(* IEC 61131-3 sources: RL_MAR/experiments/comparison/llm4plc/results/gpt-4o-mini_20260506_100619/20260506_101408, 3 files *)

(* ---- generated_code_iteration_0.st ---- *)
ructured-text
FUNCTION_BLOCK FB_SplitNumber
VAR_INPUT
    InputNumber : INT;
END_VAR

VAR_OUTPUT
    Thousands : INT;
    Hundreds : INT;
    Tens : INT;
    Ones : INT;
    Min : INT;
    error : BOOL;
    status : WORD;
END_VAR

VAR
    state : INT; // THE STATE VARIABLE
    prevState : INT; // THE PREVIOUS STATE VARIABLE
    tempNumber : INT; // Temporary variable for processing
    minValue : INT; // Variable to track the minimum non-zero digit
END_VAR

// Initialize state
state := 0;
error := FALSE;
status := 16#0000;
Thousands := 0;
Hundreds := 0;
Tens := 0;
Ones := 0;
Min := 0;

CASE state OF
    0: // STATE 0: INITIALIZE
        // Always transition to validate input
        state := 1;

    1: // STATE 1: VALIDATE INPUT
        IF InputNumber < 0 OR InputNumber > 9999 THEN
            error := TRUE;
            status := 16#8001;
            Thousands := 0;
            Hundreds := 0;
            Tens := 0;
            Ones := 0;
            Min := 0;
            state := 4; // Transition to ERROR HANDLING
        ELSE
            error := FALSE;
            status := 16#0000;
            state := 2; // Transition to SEPARATE DIGITS
        END_IF;

    2: // STATE 2: SEPARATE DIGITS
        Thousands := InputNumber / 1000;
        Hundreds := (InputNumber MOD 1000) / 100;
        Tens := (InputNumber MOD 100) / 10;
        Ones := InputNumber MOD 10;
        Min := 0; // Initialize Min
        state := 3; // Transition to FIND MINIMUM NON-ZERO DIGIT

    3: // STATE 3: FIND MINIMUM NON-ZERO DIGIT
        minValue := 32767; // Initialize minValue to maximum possible INT value

        // Compare non-zero digits
        IF Thousands > 0 THEN
            minValue := minimal(minValue, Thousands);
        END_IF;

        IF Hundreds > 0 THEN
            minValue := minimal(minValue, Hundreds);
        END_IF;

        IF Tens > 0 THEN
            minValue := minimal(minValue, Tens);
        END_IF;

        IF Ones > 0 THEN
            minValue := minimal(minValue, Ones);
        END_IF;

        // Set Min based on minValue
        IF minValue = 32767 THEN
            Min := 0; // All digits were zero
        ELSE
            Min := minValue; // Found minimum non-zero digit
        END_IF;

        state := 0; // Transition back to INITIALIZE

    4: // STATE 4: ERROR HANDLING
        // Error state already handled in STATE 1
        state := 0; // Transition back to INITIALIZE
END_CASE;

END_FUNCTION_BLOCK

(* ---- generated_code_iteration_1.st ---- *)
START_REASON
The errors in the original Structured Text (ST) code were primarily due to the incorrect handling of variable declarations and the use of the variable name "Min." In ST, "Min" is a reserved keyword in some contexts, which can lead to unexpected behavior or compilation errors. To resolve this, I will rename the variable "Min" to "MinimumValue" to avoid any conflicts. Additionally, I will ensure that the variable sections are correctly closed with "END_VAR" as required.
END_REASON

START_ST
FUNCTION_BLOCK FB_SplitNumber
VAR_INPUT
    InputNumber : INT;
END_VAR

VAR_OUTPUT
    Thousands : INT;
    Hundreds : INT;
    Tens : INT;
    Ones : INT;
    MinimumValue : INT; // Renamed from Min to MinimumValue
    error : BOOL;
    status : WORD;
END_VAR

VAR
    state : INT; // THE STATE VARIABLE
    prevState : INT; // THE PREVIOUS STATE VARIABLE
    tempNumber : INT; // Temporary variable for processing
    minValue : INT; // Variable to track the minimum non-zero digit
END_VAR

// Initialize state
state := 0;
error := FALSE;
status := 16#0000;
Thousands := 0;
Hundreds := 0;
Tens := 0;
Ones := 0;
MinimumValue := 0; // Initialize MinimumValue

CASE state OF
    0: // STATE 0: INITIALIZE
        // Always transition to validate input
        state := 1;

    1: // STATE 1: VALIDATE INPUT
        IF InputNumber < 0 OR InputNumber > 9999 THEN
            error := TRUE;
            status := 16#8001;
            Thousands := 0;
            Hundreds := 0;
            Tens := 0;
            Ones := 0;
            MinimumValue := 0; // Set MinimumValue to 0 on error
            state := 4; // Transition to ERROR HANDLING
        ELSE
            error := FALSE;
            status := 16#0000;
            state := 2; // Transition to SEPARATE DIGITS
        END_IF;

    2: // STATE 2: SEPARATE DIGITS
        Thousands := InputNumber / 1000;
        Hundreds := (InputNumber MOD 1000) / 100;
        Tens := (InputNumber MOD 100) / 10;
        Ones := InputNumber MOD 10;
        MinimumValue := 0; // Initialize MinimumValue
        state := 3; // Transition to FIND MINIMUM NON-ZERO DIGIT

    3: // STATE 3: FIND MINIMUM NON-ZERO DIGIT
        minValue := 32767; // Initialize minValue to maximum possible INT value

        // Compare non-zero digits
        IF Thousands > 0 THEN
            minValue := minimal(minValue, Thousands);
        END_IF;

        IF Hundreds > 0 THEN
            minValue := minimal(minValue, Hundreds);
        END_IF;

        IF Tens > 0 THEN
            minValue := minimal(minValue, Tens);
        END_IF;

        IF Ones > 0 THEN
            minValue := minimal(minValue, Ones);
        END_IF;

        // Set MinimumValue based on minValue
        IF minValue = 32767 THEN
            MinimumValue := 0; // All digits were zero
        ELSE
            MinimumValue := minValue; // Found minimum non-zero digit
        END_IF;

        state := 0; // Transition back to INITIALIZE

    4: // STATE 4: ERROR HANDLING
        // Error state already handled in STATE 1
        state := 0; // Transition back to INITIALIZE
END_CASE;

END_FUNCTION_BLOCK
END_ST

(* ---- generated_code_iteration_2.st ---- *)
START_REASON
The errors in the original Structured Text (ST) code were primarily due to the incorrect use of the function "minimal." In Structured Text, there is no built-in function named "minimal" for comparing values. Instead, I should use a conditional statement to determine the minimum value among the digits. I will replace the usage of "minimal" with appropriate conditional checks to find the minimum non-zero digit. Additionally, I will ensure that the variable sections are correctly closed with "END_VAR" as required.
END_REASON

START_ST
FUNCTION_BLOCK FB_SplitNumber
VAR_INPUT
    InputNumber : INT;
END_VAR

VAR_OUTPUT
    Thousands : INT;
    Hundreds : INT;
    Tens : INT;
    Ones : INT;
    MinimumValue : INT; // Renamed from Min to MinimumValue
    error : BOOL;
    status : WORD;
END_VAR

VAR
    state : INT; // THE STATE VARIABLE
    prevState : INT; // THE PREVIOUS STATE VARIABLE
    tempNumber : INT; // Temporary variable for processing
    minValue : INT; // Variable to track the minimum non-zero digit
END_VAR

// Initialize state
state := 0;
error := FALSE;
status := 16#0000;
Thousands := 0;
Hundreds := 0;
Tens := 0;
Ones := 0;
MinimumValue := 0; // Initialize MinimumValue

CASE state OF
    0: // STATE 0: INITIALIZE
        // Always transition to validate input
        state := 1;

    1: // STATE 1: VALIDATE INPUT
        IF InputNumber < 0 OR InputNumber > 9999 THEN
            error := TRUE;
            status := 16#8001;
            Thousands := 0;
            Hundreds := 0;
            Tens := 0;
            Ones := 0;
            MinimumValue := 0; // Set MinimumValue to 0 on error
            state := 4; // Transition to ERROR HANDLING
        ELSE
            error := FALSE;
            status := 16#0000;
            state := 2; // Transition to SEPARATE DIGITS
        END_IF;

    2: // STATE 2: SEPARATE DIGITS
        Thousands := InputNumber / 1000;
        Hundreds := (InputNumber MOD 1000) / 100;
        Tens := (InputNumber MOD 100) / 10;
        Ones := InputNumber MOD 10;
        MinimumValue := 0; // Initialize MinimumValue
        state := 3; // Transition to FIND MINIMUM NON-ZERO DIGIT

    3: // STATE 3: FIND MINIMUM NON-ZERO DIGIT
        minValue := 32767; // Initialize minValue to maximum possible INT value

        // Compare non-zero digits
        IF Thousands > 0 AND Thousands < minValue THEN
            minValue := Thousands;
        END_IF;

        IF Hundreds > 0 AND Hundreds < minValue THEN
            minValue := Hundreds;
        END_IF;

        IF Tens > 0 AND Tens < minValue THEN
            minValue := Tens;
        END_IF;

        IF Ones > 0 AND Ones < minValue THEN
            minValue := Ones;
        END_IF;

        // Set MinimumValue based on minValue
        IF minValue = 32767 THEN
            MinimumValue := 0; // All digits were zero
        ELSE
            MinimumValue := minValue; // Found minimum non-zero digit
        END_IF;

        state := 0; // Transition back to INITIALIZE

    4: // STATE 4: ERROR HANDLING
        // Error state already handled in STATE 1
        state := 0; // Transition back to INITIALIZE
END_CASE;

END_FUNCTION_BLOCK
END_ST
